Staubli VAL3: alreadyExist.pgx

program alreadyExist(string& x_sName[], bool& x_bFound[])
  local num l_nResult
  local string l_sMessage
  local string l_sMessage2
  local InstrItem l_iItem
begin
  switch nViewMode
    case 0
      l_iItem.sType="OUT"
    break
    case 1
      l_iItem.sType="IN"
    break
    case 2
      l_iItem.sType="NUM"
    break
  endSwitch
  // set the data
  l_iItem.sData=x_sName
  // search inside all the program - trajectory - tcp
  call prog:findItem(l_iItem,l_nResult,true)
  if l_nResult!=0
    // show the item if it exists
    call showExist(x_sName,sMessage)
    x_bFound=true
  else
    x_bFound=false
  endIf
end
